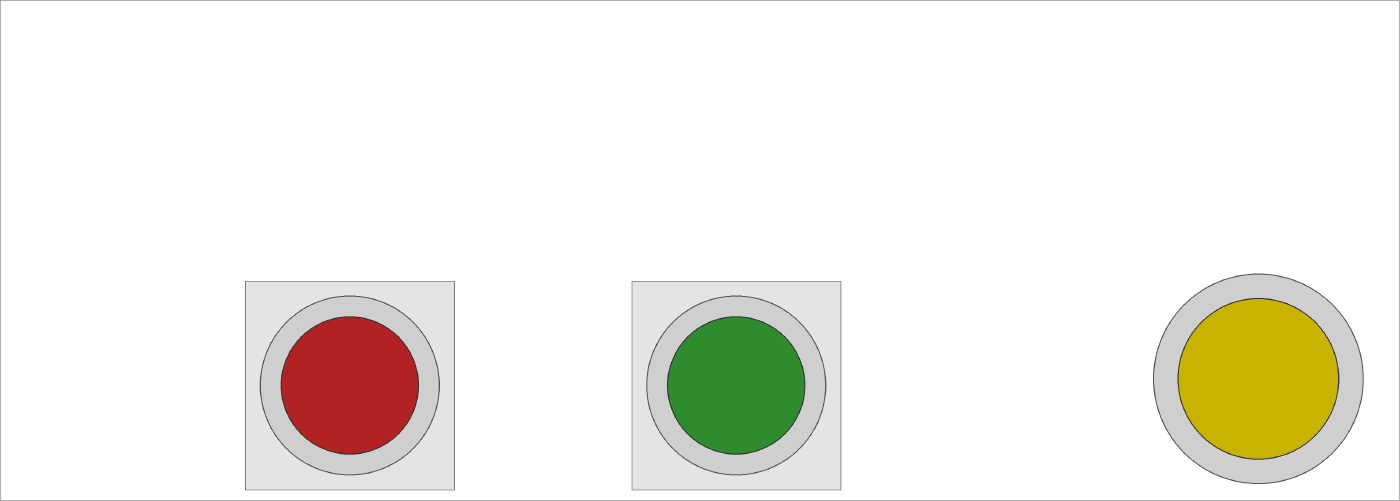
VISUALIZATION Visualization  // 1913x685
    Lamp1 (1526,351 387x334), variable: MAIN.bMotor, style: Lamp-Lamp1-Yellow
    PushSwitch (269,384 418x286), variable: MAIN.bStopButton, behaviour: TOGGLE, style: Switch-PushSwitch-Red
    PushSwitch (797,384 418x286), variable: MAIN.bStartButton, behaviour: TOGGLE, style: Switch-PushSwitch-Green
END_VISUALIZATION

(* stored: Version 1.1.0.1
   Visu Visualization: Id {b340f20a-eb51-40ef-9665-9e008c5912be} *)
